//==================================================================================================
//							Beckhoff Automation Poland
//									30.03.2017
//			Funkcja skalujaca
// 	v1.0	|| TC v 3.1.4020.32		|| - pierwsza wersja
//==================================================================================================
FUNCTION F_ScaleLREAL: LREAL
VAR_INPUT
	lrValue									: LREAL;				// Zmienna skalowana
	lrXmin									: LREAL;				// Dolny zakres zmiennej przeskalowanej
	lrXmax									: LREAL;				// Gorny zakres zmiennej przeskalowanej
	lrYmin									: LREAL;				// Dolny zakres zmiennej skalowanej
	lrYmax									: LREAL;				// Gorny zakres zmiennej skalowanej
	bLimits									: BOOL;					// Ogranicz wyjscie w przedziale lrYmin : lrYmax
END_VAR
VAR
	lrfA									: LREAL;				// Wspolczynnik kierunkowy prostej
	lrfB									: LREAL;				// Wspolczynnik przesuniecia prostej
END_VAR

IF (((lrXmax - lrXmin) < 0.01) AND ((lrXmax - lrXmin) > -0.01)) THEN
	F_ScaleLREAL := lrYmin;
ELSE
	lrfA := (lrYmax - lrYmin) / (lrXmax - lrXmin);
	lrfB := lrYmax - lrfA * lrXmax;
	F_ScaleLREAL := lrfA * lrValue + lrfB;
END_IF;
// LIMITY - opcja
IF bLimits THEN
	IF lrYmin < lrYmax THEN
		F_ScaleLREAL := LIMIT(lrYmin, F_ScaleLREAL, lrYmax);
	ELSE
		F_ScaleLREAL := LIMIT(lrYmax, F_ScaleLREAL, lrYmin);		
	END_IF	
END_IF

END_FUNCTION

(* stored: Version 1.1.0.1, ProductVersion 3.1.4026.13, FileIdentifier 51a07a25d15722a5458729987f7636082bcebde5, FileSignature 6d5683a192c3eab24eda955d3fb1574b4277f922699b4514add4105a029dab3afc06a58adb93eb6fbe5c3a8a7e1aefb011e4449fe5631c1e89bf3053e7e71fbf9a11c6341efe4cf81c6188cab840d8b90c971dda3b049d95e89351e6f6e90ccc1ef0b2892ef43c32c7454363519f8f9aacb7ea5dd13cfbd06272800a538ea99b1b185be78a7983c33f84a23e0b52f66132f7797eb43fda71872c7da9e4b5c245c1a85119706d84fa140018853eab930ea7c0998ffb3faf1cc68fe0a3de90c16e1d16c4008526d236403e88ba4b3f44ceee30eee7da9b40512fa535963a7a625493526f8133b2e0b8fa0d8de2dac3be0b1f213ee72034ee0b3dc685c7419394a2
   POU F_ScaleLREAL: Id {879b22d9-204f-4243-bfa7-bfc6d51a4a36}, SpecialFunc None *)
